(* IEC 61131-3 sources: Lasal/CPU_5344_V01/Class/ScalePotMeter, 1 file *)

(* ---- ScalePotMeter.st ---- *)
(*!
<Class
	Name               = "ScalePotMeter"
	Revision           = "0.0"
	RealtimeTask       = "false"
	CyclicTask         = "false"
	BackgroundTask     = "false"
	Sigmatek           = "false"
	OSInterface        = "false"
	HighPriority       = "false"
	Automatic          = "false"
	UpdateMode         = "Prescan"
	SharedCommandTable = "true"
	Objectsize         = "(420,240)">
	<Channels>
		<Server Name="ClassSvr" Visualized="true" Initialize="false" WriteProtected="true" Retentive="false"/>
		<Server Name="Offset" Visualized="true" Initialize="false" WriteProtected="false" Retentive="SRam"/>
		<Client Name="Dif" Required="true" Internal="false"/>
		<Client Name="Mul" Required="true" Internal="false"/>
		<Client Name="Raw" Required="true" Internal="false"/>
	</Channels>
</Class>
*)
ScalePotMeter : CLASS
  //Servers:
	ClassSvr 	: SvrChCmd_DINT;
	Offset 	: SvrCh_DINT;
  //Clients:
	Mul 	: CltCh_DINT;
	Dif 	: CltCh_DINT;
	Raw 	: CltCh_DINT;
  //Variables:
		var1 	: DINT;
		var2 	: DINT;
  //Functions:

	FUNCTION VIRTUAL GLOBAL ClassSvr::Read
		VAR_OUTPUT
			output (EAX) 	: DINT;
		END_VAR;
  //Tables:
	FUNCTION @STD
		VAR_OUTPUT
			ret_code	: CONFSTATES;
		END_VAR;
	FUNCTION GLOBAL TAB @CT_;
END_CLASS;

FUNCTION VIRTUAL GLOBAL ScalePotMeter::ClassSvr::Read
	VAR_OUTPUT
		output (EAX) 	: DINT;
	END_VAR

  Mul := Mul.Read();
  Dif := Dif.Read();
  Offset := Offset.Read();
  Raw := Raw.Read();
  if dif <> 0 then
    var1 :=raw *mul;
    var2 :=var1/dif;
    ClassSvr :=var2 +Offset;
    //ClassSvr := (raw *(mul/dif)) + offset;
  else
    ClassSvr := -99999999;
  end_if;
	output := ClassSvr;

END_FUNCTION
